// TIA Portal V18 export
// export: Created 2026-06-08T16:32:19.3539255Z, ExportSetting WithDefaults, DisplayName Totally Integrated Automation Portal, DisplayVersion V18, DisplayName TIA Portal Openness, DisplayVersion V18, DisplayName TIA Portal Version Control Interface, DisplayVersion V18, DisplayName STEP 7 Professional, DisplayVersion V18, DisplayName STEP 7 Safety, DisplayVersion V18, DisplayName WinCC Professional, DisplayVersion V18
VAR_GLOBAL   // PLC tag table "base_feeding_station"
   lid_detection AT %I0.0 : Bool;
   stop_beginning_lid_sensor AT %I0.1 : Bool;
   start_LID_feeding_convyer AT %I0.2 : Bool;
   LID_detected_grip AT %I0.3 : Bool;
   stop_LID_Feeding AT %I0.4 : Bool;
   LID_machining_entrance_sensor AT %I0.5 : Bool;
   base_Raw_counter_start AT %I0.6 : Bool;
   stop_base_begininning_convyr AT %I0.7 : Bool;
   base_gripper_detected AT %I1.0 : Bool;
   start_base_raw_feeding AT %I1.1 : Bool;
   stop_base_raw_feeding AT %I1.2 : Bool;
   stop_base_machining_convyr AT %I1.3 : Bool;
   lid_start_button AT %I1.4 : Bool;
   lid_stop_button AT %I1.5 : Bool;
   lid_emergency_button AT %I1.6 : Bool;
   base_start_button AT %I1.7 : Bool;
   base_stop_button AT %I2.0 : Bool;
   base_emergency AT %I2.1 : Bool;
   Lid_beginning_conveyr AT %Q0.0 : Bool;
   lid_feeding_conveyr AT %Q0.1 : Bool;
   Lid_pickup_x_axis AT %Q0.3 : Bool;
   lid_pickup_z_axis AT %Q0.4 : Bool;
   lid_sucction_gripper AT %Q0.5 : Bool;
   base_beginning_conveyr AT %Q0.6 : Bool;
   "lid-machinning_conveyr" AT %Q0.2 : Bool;
   base_raw_feeding_conveyr AT %Q0.7 : Bool;
   base_to_machinning_conveyr AT %Q1.0 : Bool;
   base_pickup_x_axis AT %Q1.1 : Bool;
   base_pickup_z_axis AT %Q1.2 : Bool;
   base_sucction_gripper AT %Q1.3 : Bool;
   base_start_button_1_light AT %Q1.4 : Bool;
   base_stop_button_1_light AT %Q1.5 : Bool;
   lid_start_light AT %Q1.6 : Bool;
   lid_stop_button_1_light AT %Q1.7 : Bool;
   base_raw_material AT %Q2.0 : Bool;
   lid_raw_emit AT %Q2.1 : Bool;
   state_of_start_base AT %M0.0 : Bool;
   state_of_start_LID AT %M0.1 : Bool;
   state_of_lid AT %M0.2 : Bool;
   dummy AT %M0.3 : Bool;
   To_emit_lid AT %M0.4 : Bool;
   item_ready_to_picked AT %M0.5 : Bool;
   movin_lid_z_mem AT %M0.6 : Bool;
   LID_moving_z_sensor AT %I2.4 : Bool;
   LID_moving_x_sensor AT %I2.5 : Bool;
   "dummy(1)" AT %M0.7 : Bool;
   "dummy(2)" AT %M1.0 : Bool;
   lid_belt_convyer_excess AT %Q2.2 : Bool;
   push_excess_blue_lid AT %Q2.3 : Bool;
   push_excess_green_lid AT %Q2.4 : Bool;
   Blue_vision_lid AT %I2.6 : Bool;
   green_vision_lid AT %I2.7 : Bool;
   front_blue_push_lid AT %I3.0 : Bool;
   back_blue_push_lid AT %I3.1 : Bool;
   front_green_push_lid AT %I3.2 : Bool;
   back_green_push_lid AT %I3.3 : Bool;
   into_cnc_lid_sensor AT %I3.4 : Bool;
   CNC_lid_empty AT %M1.1 : Bool;
   ONE_OBJECT_IN AT %Q2.5 : Bool;
   KEEP_DISTANCE AT %Q2.6 : Bool;
   ARE_WE_THERE_YET_BLUE_lid AT %M1.2 : Bool;
   ARE_WE_THERE_YET_GREEN_lid AT %M1.3 : Bool;
   LID_COUNTER_RESET_BUTTON_BLUE AT %I3.5 : Bool;
   TO_STORAGE_BLUE_CONVYER_lid AT %Q2.7 : Bool;
   TO_STORAGE_GREEN_CONVYER_lid AT %Q3.0 : Bool;
   TO_STORAGE_BLUE_SENSOR_lid AT %I3.6 : Bool;
   TO_STORAGE_GREEN_SENSOR_lid AT %I3.7 : Bool;
   LID_COUNTER_RESET_BUTTON_GREEN AT %I4.0 : Bool;
   "GREEN_LID_PUSHER_SORTING(FRONT LIMIT)" AT %I4.1 : Bool;
   "GREEN_LID_PUSHER_SORTING(BACK LIMITT)" AT %I4.2 : Bool;
   "BLUE_LID_PUSHER_SORTING(FRONT LIMIT)" AT %I4.3 : Bool;
   "BLUE_LID_PUSHER_SORTING(BACK LIMIT)" AT %I4.4 : Bool;
   BEGIN_SORTING_STATION_LIDS AT %I4.5 : Bool;
   BLUE_LID_VISION_SORTING AT %I4.6 : Bool;
   GREEN_LID_VISION_SORTING AT %I4.7 : Bool;
   SORTING_CONVYER_LID AT %Q3.1 : Bool;
   GREEN_LID_PUSHER_SORTING AT %Q3.2 : Bool;
   BLUE_LID_PUSHER_SORTING AT %Q3.3 : Bool;
   CNC_base_empty AT %M2.5 : Bool;
   to_emit_base AT %M1.5 : Bool;
   base_into_cnc AT %I5.0 : Bool;
   BASE_MOVE_X_SENSOR AT %I5.1 : Bool;
   BASE_MOVE_Z_SENSOR AT %I5.2 : Bool;
   DUMMY1 AT %M1.6 : Bool;
   DUMMY2 AT %M1.7 : Bool;
   DUMMY3 AT %M2.0 : Bool;
   DUMMY4 AT %M2.1 : Bool;
   DUMMY5 AT %M2.2 : Bool;
   BASE_RAW_EXESS_CONV AT %Q3.4 : Bool;
   Are_we_there_base_raw_blue AT %M2.3 : Bool;
   Are_we_there_base_raw_green AT %M2.4 : Bool;
   base_raw_blue_exes_vision AT %I5.3 : Bool;
   base_raw_green_exes_vision AT %I5.4 : Bool;
   to_blue_base_raw_storage_sensor AT %I5.5 : Bool;
   to_green_base_raw_storage_sensor AT %I5.6 : Bool;
   "push_ex_green_base raw(front)" AT %I5.7 : Bool;
   "push_ex_green_base raw (back)" AT %I6.0 : Bool;
   "pusher blue base raw (front)" AT %I6.1 : Bool;
   "pusher blue base raw (back)" AT %I6.2 : Bool;
   is_base_exsist AT %M1.4 : Bool;
   Conv_sorting_set_base AT %M2.6 : Bool;
   BEGIN_SORTING_STATION_BASE_4 AT %Q5.3 : Bool;
END_VAR
